ABB RobotStudio station: Tema2_FINAL.rspag

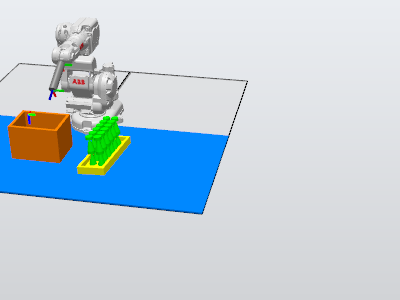
--- station ---
Station Tema2 (saved by RobotStudio 23.2.10478.1)
Controller IRB140_6_81
  mechanical unit ROB_1: IRB140_6_81_C_03, 6 joints, base frame (0, 0, 0) mm
Layout (positions relative to the parent item):
  - IRB140_6_81_C_03 [mechanism, from %ABB.RobotStudio.Models.IRB140%\IRB140_6_81_C_G_03.rslib] at (0, 0, 0) mm; joint values [0, 0, 0, 0, 0.5236, 0] (rad or m)
  - Piesa_1 [part, from Components\Piesa.rslib] at (313.39, 209.34, 232.33) mm, rotated rx 174.39 ry 1.85 rz 175.32 deg
  - Piesa_2 [part, from Components\Piesa.rslib] at (373.16, 204.45, 234.27) mm, rotated rx 174.39 ry 1.85 rz 175.32 deg
  - Piesa_3 [part, from Components\Piesa.rslib] at (432.92, 199.56, 236.2) mm, rotated rx 174.39 ry 1.85 rz 175.32 deg
  - Piesa_4 [part, from Components\Piesa.rslib] at (317.38, 218.82, 132.86) mm, rotated rx 174.39 ry 1.85 rz 175.32 deg
  - Piesa_5 [part, from Components\Piesa.rslib] at (377.15, 213.93, 134.8) mm, rotated rx 174.39 ry 1.85 rz 175.32 deg
  - Piesa_6 [part, from Components\Piesa.rslib] at (436.92, 209.04, 136.73) mm, rotated rx 174.39 ry 1.85 rz 175.32 deg
  - Piesa_7 [part, from Components\Piesa.rslib] at (492.69, 194.66, 238.14) mm, rotated rx 174.39 ry 1.85 rz 175.32 deg
  - Piesa_8 [part, from Components\Piesa.rslib] at (552.46, 189.77, 240.07) mm, rotated rx 174.39 ry 1.85 rz 175.32 deg
  - Piesa_9 [part, from Components\Piesa.rslib] at (612.23, 184.88, 242.01) mm, rotated rx 174.39 ry 1.85 rz 175.32 deg
  - Piesa_10 [part, from Components\Piesa.rslib] at (496.69, 204.14, 138.67) mm, rotated rx 174.39 ry 1.85 rz 175.32 deg
  - Piesa_11 [part, from Components\Piesa.rslib] at (556.46, 199.25, 140.6) mm, rotated rx 174.39 ry 1.85 rz 175.32 deg
  - Piesa_12 [part, from Components\Piesa.rslib] at (616.23, 194.36, 142.54) mm, rotated rx 174.39 ry 1.85 rz 175.32 deg
  - Piesa_13 [part, from Components\Piesa.rslib] at (318.07, 268.87, 238.19) mm, rotated rx 174.39 ry 1.85 rz 175.32 deg
  - Piesa_14 [part, from Components\Piesa.rslib] at (620.91, 253.89, 148.4) mm, rotated rx 174.39 ry 1.85 rz 175.32 deg
  - Piesa_15 [part, from Components\Piesa.rslib] at (377.84, 263.98, 240.13) mm, rotated rx 174.39 ry 1.85 rz 175.32 deg
  - Piesa_16 [part, from Components\Piesa.rslib] at (437.61, 259.09, 242.07) mm, rotated rx 174.39 ry 1.85 rz 175.32 deg
  - Piesa_17 [part, from Components\Piesa.rslib] at (322.07, 278.35, 138.73) mm, rotated rx 174.39 ry 1.85 rz 175.32 deg
  - Piesa_18 [part, from Components\Piesa.rslib] at (381.84, 273.46, 140.66) mm, rotated rx 174.39 ry 1.85 rz 175.32 deg
  - Piesa_19 [part, from Components\Piesa.rslib] at (441.6, 268.57, 142.6) mm, rotated rx 174.39 ry 1.85 rz 175.32 deg
  - Piesa_20 [part, from Components\Piesa.rslib] at (557.15, 249.3, 245.94) mm, rotated rx 174.39 ry 1.85 rz 175.32 deg
  - Piesa_21 [part, from Components\Piesa.rslib] at (497.38, 254.19, 244) mm, rotated rx 174.39 ry 1.85 rz 175.32 deg
  - Piesa_22 [part, from Components\Piesa.rslib] at (616.91, 244.41, 247.87) mm, rotated rx 174.39 ry 1.85 rz 175.32 deg
  - Piesa_23 [part, from Components\Piesa.rslib] at (501.37, 263.67, 144.53) mm, rotated rx 174.39 ry 1.85 rz 175.32 deg
  - Piesa_24 [part, from Components\Piesa.rslib] at (561.14, 258.78, 146.47) mm, rotated rx 174.39 ry 1.85 rz 175.32 deg
  - Cutie_preluare [part] at (-30.72, 261.88, 50) mm, size 252.6 x 340.2 x 250 mm
  - Cutie_depunere [part] at (490.45, 242.38, 41.53) mm, rotated rx 1.86 ry 5.61 rz -94.5 deg, size 185.7 x 485.7 x 50 mm
  - palet [part], size 1000 x 2000 x 10 mm
  - MyNewTool [mechanism] at (506.29, 0, 679.5) mm, rotated rx 180 ry 60 rz 180 deg
      TCP MyNewTool at (0, 0, 200) mm
      links: Part_1
Attachment: MyNewTool is attached to IRB140_6_81_C_03 / Link6
EventTableEntry 2296: ActivationMode=2, Cyclic=false, Group=, Trigger=aa_gripper 2297, Actions=[EventTableActionAttach 2298], Comment=
EventTableTriggerIO 2297: Operator=0, IOValue=[1], IRC5Controller=? -1, SignalSource=IRB140_6_81 1186
EventTableActionAttach 2298: MountObject=true, FlangeIndext=0, FindNearest=true, AttachmentParent=MyNewTool 2307, AttachmentChild=? -1, Offset=[X=1, Y=0, Z=0, W=0, X=0, Y=1, Z=0, W=0, X=0, Y=0, Z=1, W=0, X=0, Y=0, Z=0, W=1]
EventTableEntry 2311: ActivationMode=2, Cyclic=false, Group=, Trigger=aa_gripper 2312, Actions=[EventTableActionDetach 2313], Comment=
EventTableTriggerIO 2312: Operator=0, IOValue=[0], IRC5Controller=? -1, SignalSource=IRB140_6_81 1186
EventTableActionDetach 2313: AttachmentParent=MyNewTool 2307, AttachmentChild=? -1

--- Controller Data/IRB140_6_81/RAPID/TASK1/PROGMOD/CalibData.mod ---
MODULE CalibData
    PERS tooldata MyNewTool:=[TRUE,[[0,0,200],[1,0,0,0]],[1,[0,0,1],[1,0,0,0],0,0,0]];
    TASK PERS wobjdata plan_inclinat:=[FALSE,TRUE,"",[[262.764,188.299,27.226],[0.997872,0.0482292,-0.0180937,-0.0399847]],[[0,0,0],[1,0,0,0]]];
ENDMODULE

--- Controller Data/IRB140_6_81/RAPID/TASK1/PROGMOD/Module1.mod ---
MODULE Module1
        CONST robtarget home:=[[679.496732003,0,579.5],[0.5,0,0.866025404,0],[0,0,0,0],[9E+09,9E+09,9E+09,9E+09,9E+09,9E+09]];
    CONST robtarget P_pick:=[[402.235,-310.636,250],[0,0,1,0],[-1,0,-1,0],[9E+09,9E+09,9E+09,9E+09,9E+09,9E+09]];
    CONST robtarget P_place:=[[55.327278058,44.868249435,100],[0,0,1,0],[0,0,0,0],[9E+09,9E+09,9E+09,9E+09,9E+09,9E+09]];
    VAR robtarget my_pick;
    VAR robtarget my_place;
!***********************************************************
    !
    ! Module:  Module1
    !
    ! Description:
    !   <Insert description here>
    !
    ! Author: Lenovo
    !
    ! Version: 1.0
    !
    !***********************************************************


    !***********************************************************
    !
    ! Procedure main
    !
    !   This is the entry point of your program
    !
    !***********************************************************
    PROC main()
        !Add your code here

        MoveJ home,v1000,z100,MyNewTool\WObj:=wobj0;

        FOR i FROM 0 TO 23 DO
            my_pick:=offs(P_pick,(i mod 3)*70,((i div 3) mod 4)*70,-100*(i div 12));
            my_place:=offs(P_place,(i mod 6)*60,((i div 6) mod 2)*60,100*(i div 12));
            pick_and_place;
        ENDFOR

      !  FOR i FROM 12 TO 23 DO
      !      my_pick:=offs(P_pick,(i mod 3)*70,((i div 3) mod 4)*70,-100);
      !      my_place:=offs(P_place,(i mod 6)*60,((i div 6) mod 2)*60,+100);
      !  ENDFOR
        MoveL home,v1000,z100,MyNewTool\WObj:=wobj0;
    ENDPROC

    PROC pick_and_place()
        SetDO aa_gripper, 0;
        !MoveJ home,v1000,z100,MyNewTool\WObj:=wobj0;

        MoveJ offs(my_pick,0,0,200),v1000,fine,MyNewTool\WObj:=wobj0;
        MoveL my_pick,v1000,fine,MyNewTool\WObj:=wobj0;
        SetDO aa_gripper,1;
        !WaitTime 0.5;
        MoveL offs(my_pick,0,0,250),v1000,fine,MyNewTool\WObj:=wobj0;

        MoveJ offs(my_place,0,0,250),v1000,fine,MyNewTool\WObj:=plan_inclinat;
        MoveL my_place,v1000,fine,MyNewTool\WObj:=plan_inclinat;
        SetDO aa_gripper,0;
        !WaitTime 0.5;
        MoveL offs(my_place,0,0,200),v1000,fine,MyNewTool\WObj:=plan_inclinat;

        !MoveJ home,v1000,z100,MyNewTool\WObj:=wobj0;
    ENDPROC
ENDMODULE

--- Controller Data/IRB140_6_81/SYSPAR/EIO.cfg ---
EIO:CFG_1.0:6:1::
#
EIO_SIGNAL:

      -Name "aa_gripper" -SignalType "DO" -Access "All"
